(* :Description:  This function is used to convert byte structure into string text message. Structure is recived from any TCP/IP device *)
FUNCTION FUN_TcpBufferDataToString : BOOL
VAR_INPUT
	sMessageAddr		: PVOID;						(* Destination string message *)
	stReturnDataAddr	: PVOID;						(* Source TCP/IP data structure *)
END_VAR
VAR
	psMessage			: POINTER TO STRING;			(* Pointer to string converted to structure *)
	pstReturnData		: POINTER TO ST_TcpBufferData;	(* Pointer to structure made of string bytes *)
END_VAR
(*
Version history:

+-------------+------------+----------------+----------+------------------------------------------+
|Date         | Version    | created under  | Author   | Remark                                   |
+=============+============+================+==========+==========================================+
|2022-01      | 1.0.0.0    | V3.1.4024.22   | ADBO     | Function block created                   |
+-------------+------------+----------------+----------+------------------------------------------+

*)

(* Check if any input address is different than zero*)
IF sMessageAddr <> 0 AND stReturnDataAddr <> 0 THEN
	(* Access to adress*)
	psMessage := sMessageAddr;
	pstReturnData := stReturnDataAddr;
	
	(* Clear string from any old bytes *)
	MEMSET(psMessage,0,SIZEOF(psMessage^));
	
	(* Copy bytes from string to structure *)
	MEMCPY(destAddr := psMessage, srcAddr := ADR(pstReturnData^.arrData), n:= pstReturnData^.iLength);
	
	(* Function done *)	
	FUN_TcpBufferDataToString := TRUE;
(* One of adresses was not correct *)		
ELSE
	FUN_TcpBufferDataToString := FALSE;
END_IF

END_FUNCTION

(* stored: Version 1.1.0.1, ProductVersion 3.1.4024.9
   POU FUN_TcpBufferDataToString: Id {c0ea027d-9d1a-4ab2-8510-11b9b4e428b5}, SpecialFunc None *)
